INTERFACE I_QuantityLREAL EXTENDS I_Quantity


PROPERTY Val : LREAL
GET
END_GET
END_PROPERTY

END_INTERFACE

(* stored: Version 1.1.0.1
   Itf I_QuantityLREAL: Id {08c54946-8856-4097-9af1-048809742ee4}
   Property Val: Id {b2d2511a-043b-42b2-ab27-3fd7bcd93780}
   Get Get: Id {c1344037-d6a5-4916-85aa-0ca191577215} *)
